TYPE VTD_Levels_DUT :
STRUCT
	Levels_LE:	ARRAY[1..8] OF REAL;
END_STRUCT
END_TYPE

(* stored: Version 1.1.0.1
   DUT VTD_Levels_DUT: Id {5f410c75-c18e-4447-b226-6f73fd206573} *)
